{attribute 'to_string'}
TYPE E_DoorDasher_States : (
	DOOR_DASHER_DISABLED,
	DOOR_DASHER_ENABLING
	
	, DOOR_DASHER_AUTOFEED_OFF
	, DOOR_DASHER_AUTOFEED_ON
	
	, DOOR_DASHER_START
	, DOOR_DASHER_WAIT_FOR_SOURCE_TABLE_READY
	, DOOR_DASHER_WAIT_FOR_SOURCE_AND_TARGET_EXTERNAL
	, DOOR_DASHER_CENTER_DOOR_PRE_ROTATE
	, DOOR_DASHER_ROTATE_DOOR
	, DOOR_DASHER_ALIGN_DOOR
	
	, DOOR_DASHER_READY_TO_TRANSFER
	
	, DOOR_DASHER_CROSS_TRANSFER_START
	, DOOR_DASHER_CROSS_TRANSFER_ACTIVATE_CROSS_CYLS
	, DOOR_DASHER_CROSS_TRANSFER_START_SOURCE_MOTOR
	, DOOR_DASHER_CROSS_TRANSFER_FIND_SOURCE_EYE_RISING_EDGE
	, DOOR_DASHER_CROSS_TRANSFER_STOP_SOURCE_MOTOR
	, DOOR_DASHER_CROSS_TRANSFER_WAIT_FOR_ALL_DOORDASHERS_READY
	, DOOR_DASHER_CROSS_TRANSFER_START_MOTORS
	, DOOR_DASHER_CROSS_TRANSFER_FIND_TARGET_EYE_RISING_EDGE_PRE
	, DOOR_DASHER_CROSS_TRANSFER_FIND_TARGET_EYE_RISING_EDGE_POST
	, DOOR_DASHER_CROSS_TRANSFER_FIND_RISING_OR_FALLING_EDGE_OF_TARGET_EYE
	, DOOR_DASHER_CROSS_TRANSFER_STOP_MOTORS	
	, DOOR_DASHER_CROSS_TRANSFER_RESTART_TARGET_MOTOR
	, DOOR_DASHER_CROSS_TRANSFER_FIND_RISING_EDGE_OF_TARGET_FENCE_EYE
	, DOOR_DASHER_CROSS_TRANSFER_STOP_MOTORS_ON_TARGET_FENCE_EYE	
	, DOOR_DASHER_CROSS_TRANSFER_DEACTIVATE_CROSS_CYLS
	, DOOR_DASHER_CROSS_TRANSFER_ALIGN_DOOR_AT_TARGET
	, DOOR_DASHER_CROSS_TRANSFER_WAIT_FOR_ALIGN_DOOR_AT_TARGET_COMPLETE	
	, DOOR_DASHER_CROSS_TRANSFER_WAIT_FOR_ALL_DOORDASHERS_COMPLETE
	, DOOR_DASHER_CROSS_TRANSFER_COMPLETE
	
	, DOOR_DASHER_INLINE_TRANSFER_START
	, DOOR_DASHER_INLINE_TRANSFER_DEACTIVATE_CROSS_CYLS
	, DOOR_DASHER_INLINE_TRANSFER_START_SOURCE_MOTOR
	, DOOR_DASHER_INLINE_TRANSFER_FIND_SOURCE_EYE_RISING_EDGE
	, DOOR_DASHER_INLINE_TRANSFER_STOP_SOURCE_MOTOR
	, DOOR_DASHER_INLINE_TRANSFER_WAIT_FOR_ALL_DOORDASHERS_READY
	, DOOR_DASHER_INLINE_TRANSFER_START_MOTORS
	, DOOR_DASHER_INLINE_TRANSFER_FIND_TARGET_EYE_RISING_EDGE
	, DOOR_DASHER_INLINE_TRANSFER_FIND_TARGET_EYE_FALLING_EDGE
	, DOOR_DASHER_INLINE_TRANSFER_STOP_MOTORS
	, DOOR_DASHER_INLINE_TRANSFER_FEEDIN_DOOR_AT_TARGET
	, DOOR_DASHER_INLINE_TRANSFER_WAIT_FOR_FEEDIN_DOOR_AT_TARGET_COMPLETE
	, DOOR_DASHER_INLINE_TRANSFER_WAIT_FOR_ALL_DOORDASHERS_COMPLETE
	, DOOR_DASHER_INLINE_TRANSFER_COMPLETE
	
	, DOOR_DASHER_SET_SOURCE_AND_TARGET_INTERNAL
	, DOOR_DASHER_COMPLETE
	
	, DOOR_DASHER_ERROR	
);
END_TYPE

(* stored: Version 1.1.0.1, ProductVersion 3.1.4024.12
   DUT E_DoorDasher_States: Id {6afbdbbf-8a13-40a8-891a-dd2eca8ea3ec} *)
